TYPE ST_HMI_In :
STRUCT
	bStart 		:	BOOL;
	bStop 		:	BOOL;
	bAck		:	BOOL;
END_STRUCT
END_TYPE

(* stored: Version 1.1.0.1, ProductVersion 3.1.4024.12
   DUT ST_HMI_In: Id {23c941fc-32bb-4f01-b2d8-b5087f931305} *)
